FUNCTION FUN_RangeInside : BOOL
VAR_INPUT
	fValue		:LREAL;			// Actual value
	fLimitHigh	:LREAL;			// High limit for range
	fLimitLow	:LREAL;			// Low limit for range
END_VAR
VAR
	bInside		:BOOL;			// True if value is inside range
END_VAR


// Compare actual value with range
IF fValue >= fLimitLow AND fValue <= fLimitHigh THEN
	// Inside range
	bInside := TRUE;
ELSE
	// Outside of range
	bInside := FALSE;
END_IF

// Set return value
FUN_RangeInside := bInside;

END_FUNCTION

(* stored: Version 1.1.0.1, ProductVersion 3.1.4024.12
   POU FUN_RangeInside: Id {ded1f48b-970d-49da-b792-61844bbae406}, SpecialFunc None *)
